FUNCTION_BLOCK PUBLIC FB_SquareWaveGenerator
VAR_INPUT
	bStartStop : BOOL;
	tHighTime : TIME := T#1S;
	tLowTime : TIME := T#1S;
END_VAR
VAR_OUTPUT
	bOutPulse: BOOL;
END_VAR
VAR
	fbTON : TON;
	eState: (NotStarted, Started);
	bTimerState: BOOL := FALSE;
	tDuration: TIME := tHighTime;
END_VAR

fbTON (IN:= bTimerState, PT:= tDuration);

CASE eState OF
	NotStarted:
		IF bStartStop THEN
			Start();
		END_IF
		
	Started:
		IF fbTON.Q THEN
			Toggle();
		END_IF
		
		IF NOT bStartStop THEN
			Stop();
		END_IF
END_CASE

METHOD PRIVATE Start : BOOL
eState := Started;
bOutPulse := TRUE;

tDuration := tHighTime;
bTimerState := TRUE;

Start := TRUE;
END_METHOD

METHOD PRIVATE Stop : BOOL
fbTON (IN := FALSE);

bTimerState := FALSE;
eState := NotStarted;
bOutPulse := FALSE;

Stop := TRUE;
END_METHOD

METHOD PRIVATE Toggle : BOOL
fbTON (IN := FALSE);

bOutPulse := NOT bOutPulse;
IF bOutPulse THEN
	tDuration := tHighTime;
ELSE
	tDuration := tLowTime;
END_IF
bTimerState := TRUE;

Toggle := TRUE;
END_METHOD

END_FUNCTION_BLOCK

(* stored: Version 1.1.0.1, ProductVersion 3.1.4024.12
   POU FB_SquareWaveGenerator: Id {6452d076-6004-436e-b7a3-d2fccf49a044}, SpecialFunc None
   Method Start: Id {43b738a1-9377-4cc1-bbc2-828c1103e206}
   Method Stop: Id {bcb8da47-83cb-4b1a-96db-f8fa3688803e}
   Method Toggle: Id {2b07978b-68a6-4604-bc08-7ef2614c5010} *)
